Fanuc KAREL source: ko00006.KL

-- PROVISIONAL review KL for V940-1; original PC SHA256 98827c2f0c12979f7ec5bf80b4e09cdc19d203a18788e5ffc217a184ff7b1130
-- Incomplete behavior may be omitted. Consult companion uncertainty JSON. Do not deploy.
PROGRAM KO00006
%NOLOCKGROUP
-- UNRESOLVED_DECL P1 type=000101
-- UNRESOLVED_DECL P2 type=000101
-- UNRESOLVED_DECL P3 type=000101
-- UNRESOLVED_DECL P4 type=000101
-- UNRESOLVED_DECL OUT type=000102
BEGIN
  -- V9_ZERO_TABLE_METADATA_HINT layout=0001; no indexed target words; source/name/runtime held
  -- UNRESOLVED_PC offsets 5-68; opcodes 27,22,1C,22,1C,22,1C,22,1C,76,7E,4A
  -- UNRESOLVED_PC offsets 73-77; opcodes 7F
END KO00006
